// TIA Portal V19 export
DATA_BLOCK "GlobalSafetyDB"   // DB6, F_DB
{ S7_Optimized_Access := 'TRUE' }
   VAR
      GlobalEstop : Bool;
      GlobalAck : Bool;   // Used to acknowledge global failsafety
      SubordinateEstop : Bool;
      ClockByteSupervisory : Int;
   END_VAR
BEGIN
END_DATA_BLOCK
